PROGRAM P4_00_MAIN
VAR
END_VAR

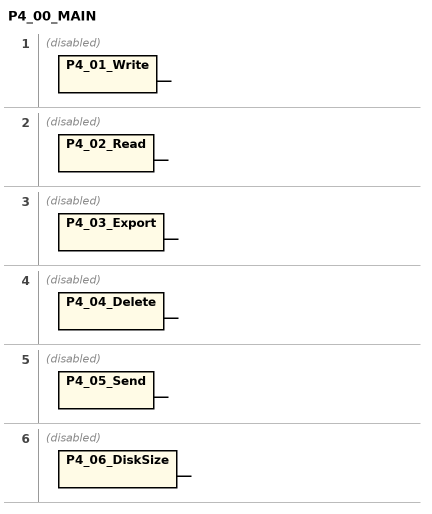
// NETWORK 1 (disabled)
// P4_01_Write();

// NETWORK 2 (disabled)
// P4_02_Read();

// NETWORK 3 (disabled)
// P4_03_Export();

// NETWORK 4 (disabled)
// P4_04_Delete();

// NETWORK 5 (disabled)
// P4_05_Send();

// NETWORK 6 (disabled)
// P4_06_DiskSize();

END_PROGRAM

(* stored: Version 1.1.0.1, ProductVersion 3.1.4026.13
   POU P4_00_MAIN: Id {d511578b-b7de-42e9-bf03-fc06d50e5046}, SpecialFunc None *)
